% RSLogix 500 project ConveyorSimulator.RSS, saved by version 8.30.00.16 %
PROJECT "UNTITLED"    % processor: MicroLogix 1000 %

PROGRAM FILES
  LAD 2 "MAIN_PROG"  8 rungs
  LAD 3 "USER_FAULT"  1 rungs
  LAD 4 "HSC_INT"  1 rungs
  LAD 5 "STI_INT"  1 rungs
  LAD 6, 7, 8, 9, 10, 11, 12, 13, 14, 15, 16: only END

DATA FILES
  O0 OUTPUT  1 elements
  I1 INPUT  2 elements
  S2 STATUS  33 elements
  B3 BINARY  32 elements
  T4 TIMER  40 elements
  C5 COUNTER  32 elements
  R6 CONTROL  16 elements
  N7 INTEGER  105 elements

LADDER 2 "MAIN_PROG"
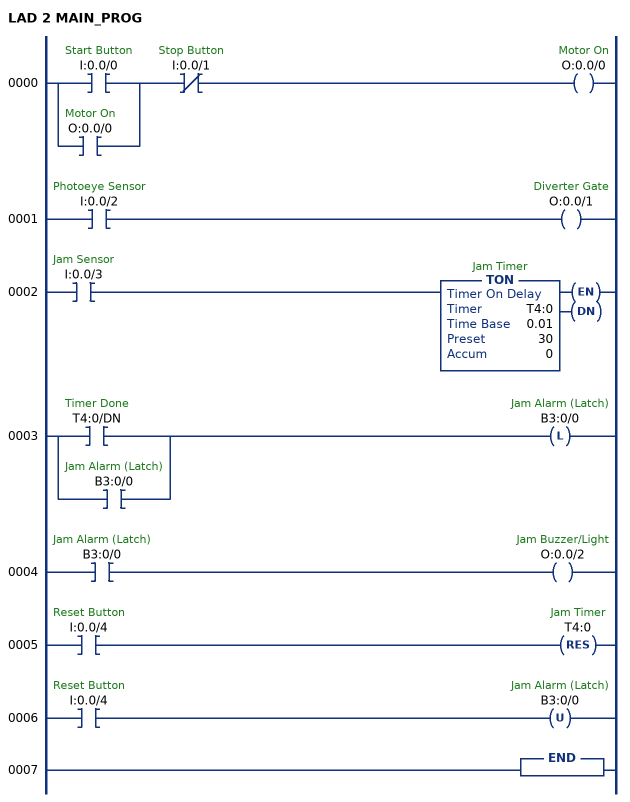
% Rung: 0 %
SOR BST XIC I:0.0/0 NXB XIC O:0.0/0 BND XIO I:0.0/1 OTE O:0.0/0 EOR
%   I:0.0/0  "Start Button" %
%   O:0.0/0  "Motor On" %
%   I:0.0/1  "Stop Button" %
% Rung: 1 %
SOR XIC I:0.0/2 OTE O:0.0/1 EOR
%   I:0.0/2  "Photoeye Sensor" %
%   O:0.0/1  "Diverter Gate" %
% Rung: 2 %
SOR XIC I:0.0/3 TON T4:0 0.01 30 0 EOR
%   I:0.0/3  "Jam Sensor" %
%   T4:0  "Jam Timer" %
% Rung: 3 %
SOR BST XIC T4:0/DN NXB XIC B3:0/0 BND OTL B3:0/0 EOR
%   T4:0/DN  "Timer Done" %
%   B3:0/0  "Jam Alarm (Latch)" %
% Rung: 4 %
SOR XIC B3:0/0 OTE O:0.0/2 EOR
%   B3:0/0  "Jam Alarm (Latch)" %
%   O:0.0/2  "Jam Buzzer/Light" %
% Rung: 5 %
SOR XIC I:0.0/4 RES T4:0 EOR
%   I:0.0/4  "Reset Button" %
%   T4:0  "Jam Timer" %
% Rung: 6 %
SOR XIC I:0.0/4 OTU B3:0/0 EOR
%   I:0.0/4  "Reset Button" %
%   B3:0/0  "Jam Alarm (Latch)" %
% Rung: 7 %
SOR END EOR

DATA TABLE (non-zero values as saved)
DATA T4
% .PRE .ACC %
% T4:0 % 30 0
